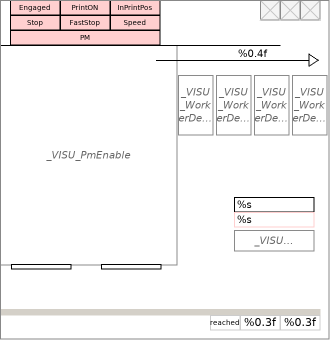
VISUALIZATION _VISU_Pm_WEU_mini  // 330x340
VAR_IN_OUT
  mInst : FB_PrintModule_WEU;
END_VAR
    Rectangle (0,60 330x280)
    RoundedRectangle (0,309 320x6), colour toggle: mInst.fbView.bMovingInd
    Frame (0,45 177x220)
        shows _VISU_PmEnable(mInst := mInst)
        p2738717112: mInst.fbView.zPos_PM
    RoundedRectangle (11,264 60x5), colour toggle: mInst.fbView.bPrintInd[2]
        p2738717112: mInst.fbView.zPos_PM
    RoundedRectangle (101,264 60x5), colour toggle: mInst.fbView.bPrintInd[1]
        p2738717112: mInst.fbView.zPos_PM
    Line (0,45) (280,45)
    Frame (254,75 35x60)
        shows _VISU_WorkerDefGrid_small(m_Inst := mInst.fbWorkerDeformation)
    Frame (292,75 35x60)
        shows _VISU_WorkerDefGrid_small(m_Inst := mInst.fbWorkerCamera)
    Frame (178,75 35x60)
        shows _VISU_WorkerDefGrid_small(m_Inst := mInst.fbWorkerPrint[2])
    Frame (216,75 35x60)
        shows _VISU_WorkerDefGrid_small(m_Inst := mInst.fbWorkerPrint[1])
    Frame (234,230 80x21)
        shows _VISU_MarkDetection_Trigger(mInst := mInst.fbMarkCameraWeu.fbMarkDetection)
    Rectangle (234,197 80x15), "%s", tooltip "active camera device", text variable: mInst.fbWorkerCamera._iActiveCam.sName
    Rectangle (234,212 80x15), "%s", tooltip "active camera mode", text variable: mInst.fbWorkerCamera._iActiveCam.eCameraMode, colour toggle: mInst.fbWorkerCamera._bCamValid
    Rectangle (235,46 80x15), "%0.4f", tooltip "PM position", text variable: mInst._fPmDistToMasterRefPos
        OnMouseClick: write the text variable via Default
    Polyline (156,60) (309,60) (309,54) (318,60) (309,66) (309,60)
    RoundedRectangle (10,30 150x15), "PM", colour toggle: mInst.fbAdsPm.stAds.bI_Enable
    RoundedRectangle (10,0 50x15), "Engaged", colour toggle: mInst._pModuleMachineState^.bEngaged
    RoundedRectangle (60,0 50x15), "PrintON", colour toggle: mInst._pModuleMachineState^.bPrintActivated
    RoundedRectangle (110,0 50x15), "InPrintPos", colour toggle: mInst._pModuleMachineState^.bUnitInPrintPosition
    RoundedRectangle (10,15 50x15), "Stop", colour toggle: NOT mInst._pModuleMachineState^.bStopRequest
    RoundedRectangle (60,15 50x15), "FastStop", colour toggle: NOT mInst._pModuleMachineState^.bFastStopRequest
    RoundedRectangle (110,15 50x15), "Speed", colour toggle: mInst.bSpeedReachedForPrinting
    RoundedRectangle (280,315 40x15), "%0.3f", tooltip "Target speed", text variable: mInst._pModuleMachineState^.fTargetSpeed
    RoundedRectangle (240,315 40x15), "%0.3f", tooltip "Current Speed", text variable: mInst.fSpeed
    RoundedRectangle (210,315 30x15), "reached", tooltip "Target speed reached", colour toggle: mInst._pModuleMachineState^.bTargetSpeedReached
    Image (260,0 20x20), invisible if: NOT mInst._pModuleMachineState^.bSleep, image: ImagePool_Steinemann.sleep_icon
    Image (280,0 20x20), invisible if: NOT mInst._pModuleMachineState^.bShutdown, image: ImagePool_Steinemann.shutdown_icon
    Image (300,0 20x20), invisible if: NOT mInst._pModuleMachineState^.bEStop, image: ImagePool_Steinemann.estop_icon
END_VISUALIZATION

(* stored: Version 1.1.0.1, ProductVersion 3.1.4024.11
   Visu _VISU_Pm_WEU_mini: Id {89f3b72d-0459-4cd1-88bb-c78f4ac36ea9} *)
